FUNCTION_BLOCK FB_System_HS_231
VAR_INPUT
	Freigabe_auto			: BOOL;
	Betrieb_Anford_auto		: BOOL;
	Regelung_Modus_auto		: SINT;
END_VAR
VAR_OUTPUT
	{attribute 'OPC.UA.DA' := '1'}Parameter					: ST_System_HS_Parameter;	
	{attribute 'OPC.UA.DA' := '1'}Steuerung					: ST_System_HS_Steuerung;	
	{attribute 'OPC.UA.DA' := '1'}Zustand						: ST_System_HS_Zustand;	
END_VAR
VAR
	Heizstaebe_231_WW			: FB_HS;
	Regelung					: FB_System_HS_Regelung;
	Zustandscheck				: FB_System_HS_Zustandscheck;
	Logik						: FB_System_HS_Logik;
	Sollwertscheck				: FB_System_HS_Sollwertscheck;
END_VAR

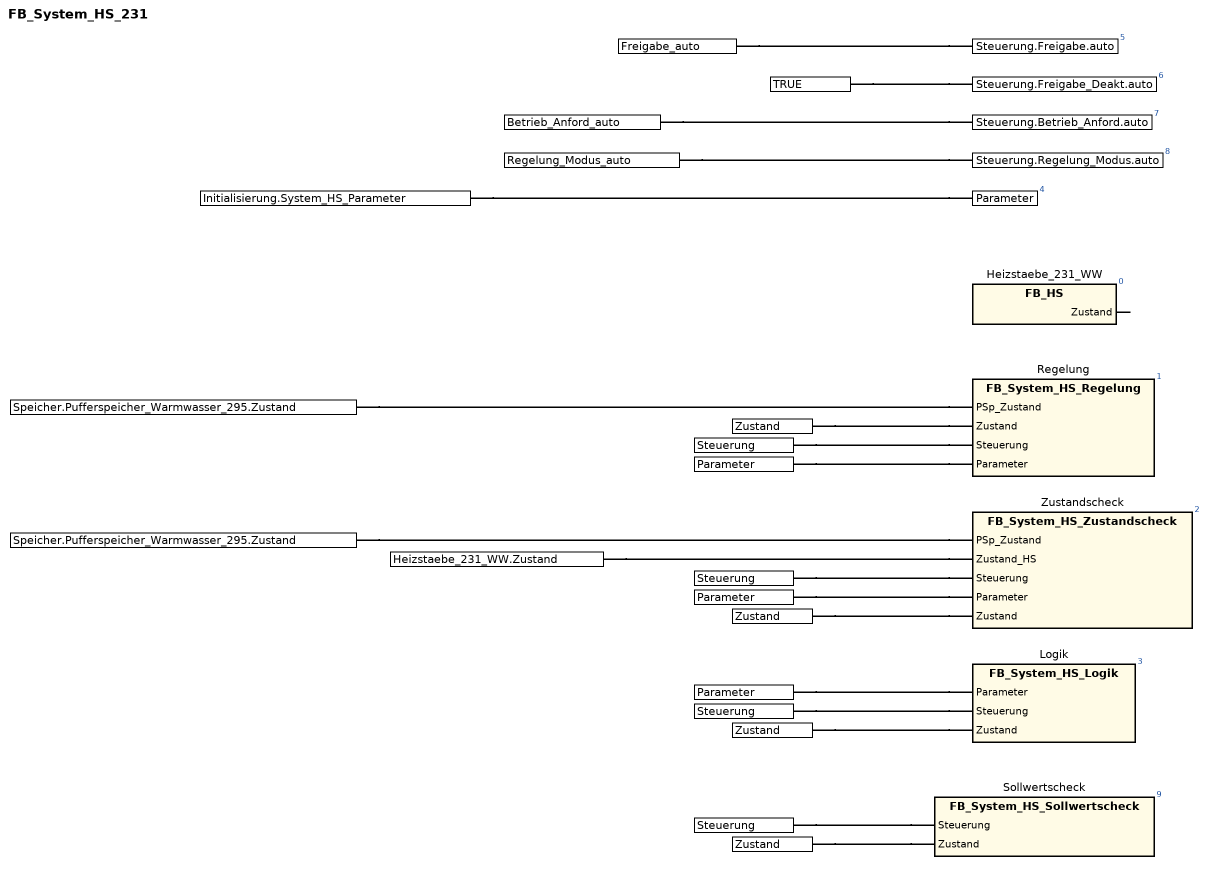
Heizstaebe_231_WW(); // FB_HS
Regelung(
    PSp_Zustand := Speicher.Pufferspeicher_Warmwasser_295.Zustand,
    Zustand := Zustand,
    Steuerung := Steuerung,
    Parameter := Parameter); // FB_System_HS_Regelung
Zustandscheck(
    PSp_Zustand := Speicher.Pufferspeicher_Warmwasser_295.Zustand,
    Zustand_HS := Heizstaebe_231_WW.Zustand,
    Steuerung := Steuerung,
    Parameter := Parameter,
    Zustand := Zustand); // FB_System_HS_Zustandscheck
Logik(Parameter := Parameter, Steuerung := Steuerung, Zustand := Zustand); // FB_System_HS_Logik
Parameter := Initialisierung.System_HS_Parameter;
Steuerung.Freigabe.auto := Freigabe_auto;
Steuerung.Freigabe_Deakt.auto := TRUE;
Steuerung.Betrieb_Anford.auto := Betrieb_Anford_auto;
Steuerung.Regelung_Modus.auto := Regelung_Modus_auto;
Sollwertscheck(Steuerung := Steuerung, Zustand := Zustand); // FB_System_HS_Sollwertscheck

END_FUNCTION_BLOCK

(* stored: Version 1.1.0.1, ProductVersion 3.1.4024.9
   POU FB_System_HS_231: Id {8fafa384-19b9-4668-a804-e04c6d956d7b}, SpecialFunc None *)
